# EPICS substitutions: iocs/linkamIOC/linkamApp/Db/linkam.substitutions
# Macros:
#  P        PV Prefix for Linkam temp. controller
#  PORT     Asyn PORT
#  ADDR     Asyn ADDR
#  TIMEOUT  Asyn TIMEOUT
#  name     Template argument
file $(LINKAM3)/db/Linkam.template
{
pattern { P, PORT, ADDR, TIMEOUT, name }
    { "EA-LINKAM-01", "EA-LINKAM-01_AP", "0", "1", "LINKAM1" }
}
